FUNCTION_BLOCK FB_SaMElementAbort EXTENDS FB_SaMElement
VAR
END_VAR

METHOD FB_init : BOOL
VAR_INPUT
	bInitRetains : BOOL; // if TRUE, the retain variables are initialized (warm start / cold start)
	bInCopyCode : BOOL;  // if TRUE, the instance afterwards gets moved into the copy code (online change)
END_VAR
THIS^.SetText (eLocation := E_BaseLocation.pl, wsDescription := "Przerwany");
THIS^.SetText (eLocation := E_BaseLocation.en, wsDescription := "Aborted");
THIS^.SetText (eLocation := E_BaseLocation.de, wsDescription := "Abgebrochen");
THIS^.SetName (stName := THIS^.GetTexts ());
END_METHOD

END_FUNCTION_BLOCK

(* stored: Version 1.1.0.1
   POU FB_SaMElementAbort: Id {6fa8edf3-f184-0e10-37fc-291d9b868d33}, SpecialFunc None
   Method FB_init: Id {bc2e7125-3e5c-0ab4-33e2-6f88147eac86} *)
